FUNCTION_BLOCK DataPanel_xDB0808_DIO_SAE_J1939 (* Service Interface Function Block Type *)
  (* Standard: SAE J1939; Function: Combo Block: 8 Inputs/8 Outputs (includes all input/output types); Type: DP-34044-1-000; Description: Copyright (c) 2018, 2023 Jose Cabral, HR Agrartechnik GmbH This program and the accompanying materials are made available under the terms of the Eclipse Public License 2.0 which is available at https://www.eclipse.org/legal/epl-2.0/ SPDX-License-Identifier: EPL-2.0 this maps to IX/QX *)
  (* Version 1.0, 2018-12-05, Jose Cabral *)
  (* Version 1.1, 2022-08-04, Franz Höpfinger, HR Agrartechnik GmbH *)
  (* Version 1.2, 2023-01-05, Franz Höpfinger, HR Agrartechnik GmbH *)
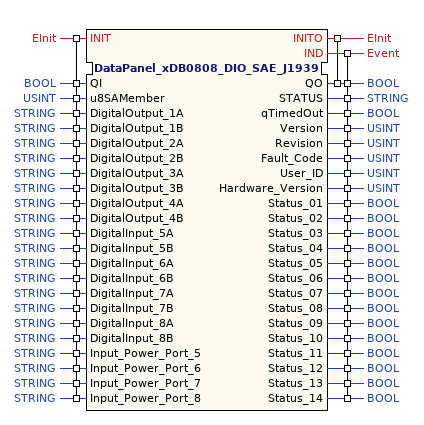
  EVENT_INPUT
    INIT : EInit WITH QI, u8SAMember, DigitalOutput_1A, DigitalOutput_1B, DigitalOutput_2A, DigitalOutput_2B, DigitalOutput_3A, DigitalOutput_3B, DigitalOutput_4A, DigitalOutput_4B, DigitalInput_5A, DigitalInput_5B, DigitalInput_7A, DigitalInput_6A, DigitalInput_6B, DigitalInput_7B, DigitalInput_8A, DigitalInput_8B, Input_Power_Port_5, Input_Power_Port_6, Input_Power_Port_7, Input_Power_Port_8; (* Service Initialization *)
  END_EVENT
  EVENT_OUTPUT
    INITO : EInit WITH QO; (* Initialization Confirm *)
    IND WITH QO, STATUS, qTimedOut, Version, Revision, Fault_Code, User_ID, Hardware_Version, Status_01, Status_02, Status_03, Status_04, Status_05, Status_06, Status_07, Status_08, Status_09, Status_10, Status_11, Status_12, Status_13, Status_14; (* Indication from Resource *)
  END_EVENT
  VAR_INPUT
    QI : BOOL; (* Event Input Qualifier *)
    u8SAMember : USINT := MI::MI_00; (* Node SA 224..239 *)
    DigitalOutput_1A : STRING;
    DigitalOutput_1B : STRING;
    DigitalOutput_2A : STRING;
    DigitalOutput_2B : STRING;
    DigitalOutput_3A : STRING;
    DigitalOutput_3B : STRING;
    DigitalOutput_4A : STRING;
    DigitalOutput_4B : STRING;
    DigitalInput_5A : STRING;
    DigitalInput_5B : STRING;
    DigitalInput_6A : STRING;
    DigitalInput_6B : STRING;
    DigitalInput_7A : STRING;
    DigitalInput_7B : STRING;
    DigitalInput_8A : STRING;
    DigitalInput_8B : STRING;
    Input_Power_Port_5 : STRING;
    Input_Power_Port_6 : STRING;
    Input_Power_Port_7 : STRING;
    Input_Power_Port_8 : STRING;
  END_VAR
  VAR_OUTPUT
    QO : BOOL; (* Event Output Qualifier *)
    STATUS : STRING; (* Service Status *)
    qTimedOut : BOOL;
    Version : USINT;
    Revision : USINT;
    Fault_Code : USINT;
    User_ID : USINT;
    Hardware_Version : USINT;
    Status_01 : BOOL;
    Status_02 : BOOL;
    Status_03 : BOOL;
    Status_04 : BOOL;
    Status_05 : BOOL;
    Status_06 : BOOL;
    Status_07 : BOOL;
    Status_08 : BOOL;
    Status_09 : BOOL;
    Status_10 : BOOL;
    Status_11 : BOOL;
    Status_12 : BOOL;
    Status_13 : BOOL;
    Status_14 : BOOL;
  END_VAR
END_FUNCTION_BLOCK
